PROGRAM MAIN
VAR
END_VAR

myVeryFirstTcoContext.Run();

END_PROGRAM

(* stored: Version 1.1.0.1, ProductVersion 3.1.4024.11
   POU MAIN: Id {f972a0b9-bbb2-4c30-9b3e-cef96ed26ba8}, SpecialFunc None *)
